(*
SPDX-FileCopyrightText: © 2026 Oleksandr Tiutyk <trofimich@gmail.com>
SPDX-License-Identifier: MIT
License: https://opensource.org/license/mit
*)

TYPE HMI_TRAFFIC_LIGHT_STATUSES :
STRUCT
	RedLightIsActive : BOOL;	
	YellowLightIsActive : BOOL;	
	GreenLightIsActive : BOOL;	
END_STRUCT
END_TYPE

(* stored: Version 1.1.0.1
   DUT HMI_TRAFFIC_LIGHT_STATUSES: Id {418af67d-dc9f-42e8-a039-2e251c781904} *)
